VISUALIZATION Visualization  // 2x2
END_VISUALIZATION

(* stored: Version 1.1.0.1, ProductVersion 3.1.4024.15
   Visu Visualization: Id {97a726b1-c93f-49cb-8adb-dc603d80a939} *)
